// TIA Portal project "Question 1 (class assignment)" (V15)

(* hardware
DEVICE "S7-1200 station_1"  S7-1200 Station
   slot 0: "Rack_0"  S7-1200 Rack  Rack  V1.0
   slot 1: "PLC_1"  CPU 1211C DC/DC/DC  6ES7 211-1AE40-0XB0  V4.2
*)

// ===== PLC "PLC_1"  CPU 1211C DC/DC/DC =====

VAR_GLOBAL   // PLC tag table "Default tag table"
   "START" AT %I0.0 : Bool;
   "STOP" AT %I0.2 : Bool;
   "EMERGENCY" AT %I0.3 : Bool;
   "Tag_4" AT %M0.0 : Bool;
   "REF SENS1" AT %I0.4 : Bool;
   "Main Conv." AT %Q0.0 : Bool;
   "REF SENS2" AT %I0.5 : Bool;
   "CONV 1" AT %Q0.1 : Bool;
   "REF SENS3" AT %I0.6 : Bool;
   "Tag_1" AT %MW200 : Int;
   "Tag_2" AT %M0.1 : Bool;
   "CONV 2" AT %Q0.2 : Bool;
   "REF SENS4" AT %I0.7 : Bool;
   "Tag_3" AT %M0.3 : Bool;
   "Tag_5" AT %MW201 : Int;
END_VAR

// folder: System blocks/Program resources

DATA_BLOCK "TIMER_1S"   // DB1
{ S7_Optimized_Access := 'TRUE' }
AUTHOR : Simatic
FAMILY : IEC
NAME : IEC_TMR
VERSION : 1.0
// stored: InstanceOfName IEC_TIMER
"IEC_TIMER"
BEGIN
END_DATA_BLOCK

DATA_BLOCK "COUNTER_5"   // DB2
{ S7_Optimized_Access := 'TRUE' }
AUTHOR : Simatic
FAMILY : IEC
NAME : CNTR
VERSION : 1.0
// stored: InstanceOfName IEC_COUNTER
"IEC_COUNTER"
BEGIN
END_DATA_BLOCK

DATA_BLOCK "COUNTER_2"   // DB3
{ S7_Optimized_Access := 'TRUE' }
AUTHOR : Simatic
FAMILY : IEC
NAME : CNTR
VERSION : 1.0
// stored: InstanceOfName IEC_COUNTER
"IEC_COUNTER"
BEGIN
END_DATA_BLOCK

// folder: (top level)

ORGANIZATION_BLOCK "Main"   // OB1, LAD, ProgramCycle
TITLE = "Main Program Sweep (Cycle)"
{ S7_Optimized_Access := 'TRUE' }
VERSION : 0.1
   VAR_INPUT
      Initial_Call : Bool;   // Initial call of this OB
      Remanence : Bool;   // =True, if remanent data are available
   END_VAR
   VAR_TEMP
      TIMER_COUNTER : Time;
   END_VAR
BEGIN

REGION Network 1
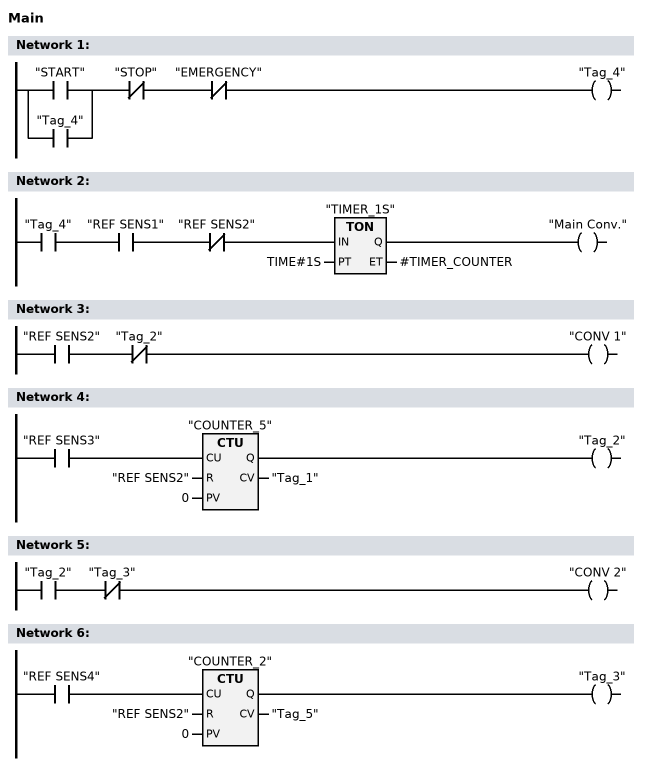
   RUNG wire#powerrail
      Contact( "START" )
      wire#w1
      I_Contact( "STOP" )
      I_Contact( "EMERGENCY" )
      Coil( "Tag_4" )
   END_RUNG
   RUNG wire#powerrail
      Contact( "Tag_4" )
   END_RUNG wire#w1
   // the same network as SCL:
   "Tag_4" := ("START" OR "Tag_4") AND NOT "STOP" AND NOT "EMERGENCY";
END_REGION

REGION Network 2
   "TIMER_1S".TON(IN := "Tag_4" AND "REF SENS1" AND NOT "REF SENS2", PT := TIME#1S, ET => #TIMER_COUNTER);
   "Main Conv." := "TIMER_1S".Q;
END_REGION

REGION Network 3
   RUNG wire#powerrail
      Contact( "REF SENS2" )
      I_Contact( "Tag_2" )
      Coil( "CONV 1" )
   END_RUNG
   // the same network as SCL:
   "CONV 1" := "REF SENS2" AND NOT "Tag_2";
END_REGION

REGION Network 4
   "COUNTER_5".CTU(CU := "REF SENS3", R := "REF SENS2", PV := 0, CV => "Tag_1");
   "Tag_2" := "COUNTER_5".Q;
END_REGION

REGION Network 5
   RUNG wire#powerrail
      Contact( "Tag_2" )
      I_Contact( "Tag_3" )
      Coil( "CONV 2" )
   END_RUNG
   // the same network as SCL:
   "CONV 2" := "Tag_2" AND NOT "Tag_3";
END_REGION

REGION Network 6
   "COUNTER_2".CTU(CU := "REF SENS4", R := "REF SENS2", PV := 0, CV => "Tag_5");
   "Tag_3" := "COUNTER_2".Q;
END_REGION
END_ORGANIZATION_BLOCK